# EPICS autosave request: apps/lakeshore450App/Db/lakeshore450_settings.req
#
# LakeShore Model 450 Gaussmeter
#
# Author: Wesley Moore
# Date:   Oct 2014
#

$(P)$(R)RANGE:SET
$(P)$(R)UNITS:SET
$(P)$(R)FIELDCOMP:SET
$(P)$(R)TEMPCOMP:SET
$(P)$(R)MODE:SET
$(P)$(R)LOCK:SET

## Restore last.  RANGE:SET will turn off auto range if changed.
$(P)$(R)AUTO_RANGE:SET
